PROGRAM MAIN
VAR
END_VAR

Process();

END_PROGRAM

(* stored: Version 1.1.0.1, ProductVersion 3.1.4024.12
   POU MAIN: Id {b2963d96-5b4d-4734-ab07-19c9ef52009d}, SpecialFunc None *)
